FUNCTION F_Sine : LREAL
VAR_INPUT
	fTime : LREAL;
END_VAR
VAR_OUTPUT
	SinuSignal : LREAL;
END_VAR
VAR

END_VAR

SinuSignal :=  0.2*SIN(2*PI*fTime/20.0); //unit [m]

END_FUNCTION

(* stored: Version 1.1.0.1, ProductVersion 3.1.4024.12
   POU F_Sine: Id {861145ac-0d3d-42b1-b1e7-c434a79e0dab}, SpecialFunc None *)
